// TIA Portal V20 export
VAR_GLOBAL   // PLC tag table "Unit1Em1_Servo"
END_VAR
